{attribute addProperty BoxType "EJ7334-0008-0016"}
{attribute addProperty Id "DCM_Status_ChannelAT %I*ARRAY[0..3] OF DCM_Status_Channel_DBE0EA1F6480DCM_Outputs_ChannelAT %Q*ARRAY[0..3] OF DCM_Outputs_Channel_1F77C8C2128160WcStateAT %I*WcState_98A4DF7520.250InfoDataAT %I*InfoData_BC63D37F80100"}
{attribute addProperty CRC "3748668872"}
{attribute addProperty SizeInBites "274"}
{attribute addProperty SizeInBytes "34.25"}
TYPE EJ7334_68079CA9 :
STRUCT
	{attribute addProperty Name "DCM_Status_Channel"}
	DCM_Status_Channel : ARRAY[0..3] OF DCM_Status_Channel_DBE0EA1F;
	{attribute addProperty Name "DCM_Outputs_Channel"}
	DCM_Outputs_Channel : ARRAY[0..3] OF DCM_Outputs_Channel_1F77C8C2;
	{attribute addProperty Name "WcState"}
	WcState : WcState_98A4DF75;
	{attribute addProperty Name "InfoData"}
	InfoData : InfoData_BC63D37F;
END_STRUCT
END_TYPE

(* stored: Version 1.2.0.0, ProductVersion 3.1.4024.9
   DUT EJ7334_68079CA9: Id {b226664b-db19-4cfd-9819-7540f5cd6dbe} *)
